// TIA Portal V19 export
FUNCTION_BLOCK "Axis_ReloadPosition_FB"   // FB32, LAD
TITLE = ENCODER RELOAD POSITION PROCEDURE
// stored: Access Published, MemoryReserve 100, SetENOAutomatically false
   VAR_INPUT
      OptionON : Bool;
      Execute : Bool;
      Rst : Bool;
      Ax_Sts_PM : "TAx_Pos_Sts";
      Ax_Sts_SIEMENS : "TAx_STATUSWORD";
   END_VAR
   VAR_OUTPUT
      Ready : Bool;
      Running : Bool;
      Done : Bool;
      AlarmsPresence : Bool;
      Ctrl_ForcePosCtrl : Bool;
      Ctrl_ReloadPosition : Bool;
      Ctrl_ReloadPosAx : LReal;
   END_VAR
   VAR_IN_OUT
      TO_Ax : TO_PositioningAxis;
      Persistent_AxisReloadPostion_OK : Bool;
      Persistent_ActualPosition : LReal;
   END_VAR
   VAR
      Status : Int;
      Alarm : Struct
         TOut_AxisHomingPermitted : Bool;
         TOut_ExecutionAxisHoming : Bool;
      END_STRUCT;
      TON_TimeOutInit : TON_TIME;
   END_VAR
BEGIN

REGION Network 1: Reset alarms
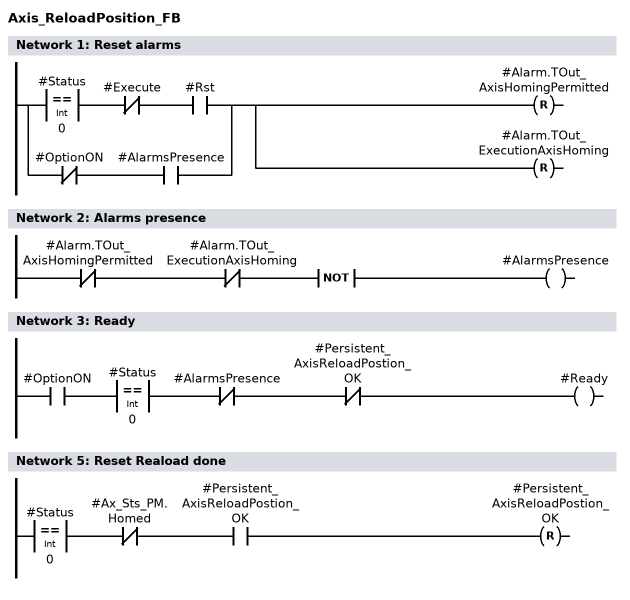
   RUNG wire#powerrail
      { S7_Templates := "SrcType := Int" } EQ_Contact(in1 := #Status, in2 := 0)
      I_Contact( #Execute )
      Contact( #Rst )
      wire#w1
      R_Coil( #Alarm.TOut_AxisHomingPermitted )
   END_RUNG
   RUNG wire#powerrail
      I_Contact( #OptionON )
      Contact( #AlarmsPresence )
   END_RUNG wire#w1
   RUNG wire#w1
      R_Coil( #Alarm.TOut_ExecutionAxisHoming )
   END_RUNG
   // the same network as SCL:
   IF ((#Status = 0) AND NOT #Execute AND #Rst) OR (NOT #OptionON AND #AlarmsPresence) THEN
       #Alarm.TOut_AxisHomingPermitted := FALSE;
       #Alarm.TOut_ExecutionAxisHoming := FALSE;
   END_IF;
END_REGION

REGION Network 2: Alarms presence
   RUNG wire#powerrail
      I_Contact( #Alarm.TOut_AxisHomingPermitted )
      I_Contact( #Alarm.TOut_ExecutionAxisHoming )
      Not()
      Coil( #AlarmsPresence )
   END_RUNG
   // the same network as SCL:
   #AlarmsPresence := NOT (NOT #Alarm.TOut_AxisHomingPermitted AND NOT #Alarm.TOut_ExecutionAxisHoming);
END_REGION

REGION Network 3: Ready
   RUNG wire#powerrail
      Contact( #OptionON )
      { S7_Templates := "SrcType := Int" } EQ_Contact(in1 := #Status, in2 := 0)
      I_Contact( #AlarmsPresence )
      I_Contact( #Persistent_AxisReloadPostion_OK )
      Coil( #Ready )
   END_RUNG
   // the same network as SCL:
   #Ready := #OptionON AND (#Status = 0) AND NOT #AlarmsPresence AND NOT #Persistent_AxisReloadPostion_OK;
END_REGION

REGION Network 4 (SCL): Sequence
   CASE #Status OF

       //=============================================================================================
       // STATUS = 0 IDLE
       //=============================================================================================
       // 

       0:

           #TON_TimeOutInit(IN:=FALSE,PT:=T#10s);

           #Ctrl_ForcePosCtrl := FALSE;

           #Ctrl_ReloadPosition := FALSE;


           #Running := FALSE;
           #Done := FALSE;


           IF  #Ready AND #Execute THEN

               #Running := TRUE;
               #Ready := FALSE;

               #Status += 1;

           END_IF;



       //=============================================================================================
       // STATUS = 1 WAIT HOMING PERMISSION THEN START COMMAND
       //=============================================================================================
       //     


       1:

           #TON_TimeOutInit(IN:=TRUE,PT:=T#10s);


           #Ctrl_ForcePosCtrl := #Ax_Sts_SIEMENS.NonPositionControlled;



           IF  #TON_TimeOutInit.Q THEN

               #Alarm.TOut_AxisHomingPermitted := TRUE;

               #Status := 0;


           ELSIF   #Ctrl_ForcePosCtrl OR #Ax_Sts_PM.Enabled  THEN

               ;

           ELSIF   #Ax_Sts_PM.HomingPermitted THEN

               #Ctrl_ReloadPosition := TRUE;


               IF #TO_Ax.Modulo.Enable THEN

                   IF #Persistent_ActualPosition >= #TO_Ax.Modulo.StartValue AND #Persistent_ActualPosition <= #TO_Ax.Modulo.Length THEN
                       #Ctrl_ReloadPosAx := #Persistent_ActualPosition;
                   ELSE
                       #Ctrl_ReloadPosAx := 0.0;
                   END_IF;
               ELSE
                   #Ctrl_ReloadPosAx := #Persistent_ActualPosition;
               END_IF;


               #Status += 1;

           END_IF;


       //=============================================================================================
       // STATUS = 2 WAIT HOMING DONE
       //=============================================================================================
       //      

       2:


           #TON_TimeOutInit(IN:=TRUE,PT:=T#10s);


           IF   #TON_TimeOutInit.Q THEN

               #Alarm.TOut_ExecutionAxisHoming := TRUE;

               #Status := 0;

           ELSIF      #Ax_Sts_PM.Homed AND #Ax_Sts_PM.HomingDone THEN



               #Status += 1;

           END_IF;



       //=============================================================================================
       // STATUS = 3 DONE
       //=============================================================================================
       //    
       3:

           #TON_TimeOutInit(IN:=FALSE,PT:=T#10s);



           #Ctrl_ReloadPosition := FALSE;

           #Ctrl_ForcePosCtrl := FALSE;


           #Persistent_AxisReloadPostion_OK := TRUE;

           #Done := TRUE;


           IF NOT #Execute THEN
               #Status := 0;
           END_IF;



       ELSE
           #Status := 0;

   END_CASE;
END_REGION

REGION Network 5: Reset Reaload done
   RUNG wire#powerrail
      { S7_Templates := "SrcType := Int" } EQ_Contact(in1 := #Status, in2 := 0)
      I_Contact( #Ax_Sts_PM.Homed )
      Contact( #Persistent_AxisReloadPostion_OK )
      R_Coil( #Persistent_AxisReloadPostion_OK )
   END_RUNG
   // the same network as SCL:
   IF (#Status = 0) AND NOT #Ax_Sts_PM.Homed AND #Persistent_AxisReloadPostion_OK THEN
       #Persistent_AxisReloadPostion_OK := FALSE;
   END_IF;
END_REGION

REGION Network 6: >
END_REGION

REGION Network 7: >
END_REGION

REGION Network 8: >
END_REGION
END_FUNCTION_BLOCK
